(* CODESYS project addition_3.xml

Project tree, tasks and I/O mapping:
  program addition_3 [ST]
*)

// addition_3
PROGRAM addition_3
VAR
	state	:INT;
END_VAR

IF TRUE = FALSE AND TRUE THEN
	state		:=		0;
END_IF

END_PROGRAM
